Staubli VAL3: Control_LeftS.pgx

public program Control_LeftS(string x_sLeftList)
  local bool l_bRes
  local string l_sBuff[20]
begin
  //在屏幕左边进行显示
  //左边的x_sLeftList 是显示的字符串数
  //字符串以,作为分割符
  call Str_SplitComma(l_bRes,x_sLeftList,l_sBuff)
  if !l_bRes
    return
  endIf

  call Control_Left(l_sBuff)
end
